FUNCTION TryConvert_LWORD_TO_TOD : BOOL
VAR_INPUT
	in : LWORD;
	out : REFERENCE TO TOD;
END_VAR

IF in > DatatypeLimits.MAX_VALUE_OF_LWORD_WHICH_CAN_BE_HELD_IN_A_TOD THEN
	RETURN;
END_IF

out := LWORD_TO_TOD(in);
TryConvert_LWORD_TO_TOD := TRUE;

END_FUNCTION

(* stored: Version 1.1.0.1, ProductVersion 3.1.4024.12
   POU TryConvert_LWORD_TO_TOD: Id {848ef5d5-0f21-4c2a-86f9-7ee72ea2a7e3}, SpecialFunc None *)
